{attribute addProperty BoxType "EL3773-0000-0016"}
{attribute addProperty Id "I2_STATUSAT %I*I2_STATUS_F9B4A013162"}
{attribute addProperty CRC "2208416549"}
{attribute addProperty SizeInBites "16"}
{attribute addProperty SizeInBytes "2"}
TYPE L2_Current_Status_83A1C325 :
STRUCT
	{attribute addProperty Name "I2_STATUS"}
	I2_STATUS AT %I* : I2_STATUS_F9B4A013;
END_STRUCT
END_TYPE

(* stored: Version 1.2.0.0, ProductVersion 3.1.4024.9
   DUT L2_Current_Status_83A1C325: Id {f13cb055-3d5b-4bd8-a805-519185b420c8} *)
